{attribute 'qualified_only'}
{attribute 'strict'}
TYPE EFeedbackMsgPolarisationFW212C :
(
	CheckConnectionMsg := 10,
    PositionMsg,
    PositionCountMsg,
    IdMsg,
    CustomMsg
);
END_TYPE

(* stored: Version 1.1.0.1, ProductVersion 3.1.4024.4
   DUT EFeedbackMsgPolarisationFW212C: Id {210c92b5-8003-4816-9793-7d4227280f8f} *)
